// TIA Portal V17 export
// export: Created 2024-08-09T12:53:10.3417679Z, ExportSetting WithDefaults, DisplayName Totally Integrated Automation Portal, DisplayVersion V17 Update 7, DisplayName TIA Portal Openness, DisplayVersion V17 Update 7, DisplayName TIA Portal Version Control Interface, DisplayVersion V17, DisplayName STEP 7 Professional, DisplayVersion V17 Update 7, DisplayName STEP 7 Safety, DisplayVersion V17 Update 6, DisplayName WinCC Professional, DisplayVersion V17 Update 7
VAR_GLOBAL   // PLC tag table "Dec_Niveaux_Rec"
END_VAR
VAR_GLOBAL CONSTANT   // user constants
   REC_Repos_Niv : USInt := 0;
   REC_AttenteAval_Niv : USInt := 15;
   REC_AttenteAmont_Niv : USInt := 30;
   REC_Lancement_Niv : USInt := 45;
   REC_Prepositionnement_Niv : USInt := 60;
   REC_AttenteCircuitPositionne_Niv : USInt := 75;
   REC_AttenteProduit_Niv : USInt := 90;
   REC_Surveillance_Niv : USInt := 105;
   REC_ChangementDestination_Niv : USInt := 120;
   REC_Suspension_Niv : USInt := 150;
   REC_TestQtePassee_Niv : USInt := 165;
   REC_AttenteAcquitNettoyage_Niv : USInt := 180;
   REC_Vidange_Niv : USInt := 195;
   REC_MajBase_Niv : USInt := 210;
   REC_FinLot_Niv : USInt := 255;
   REC_ChangementNoeud_Niv : USInt := 135;
END_VAR
